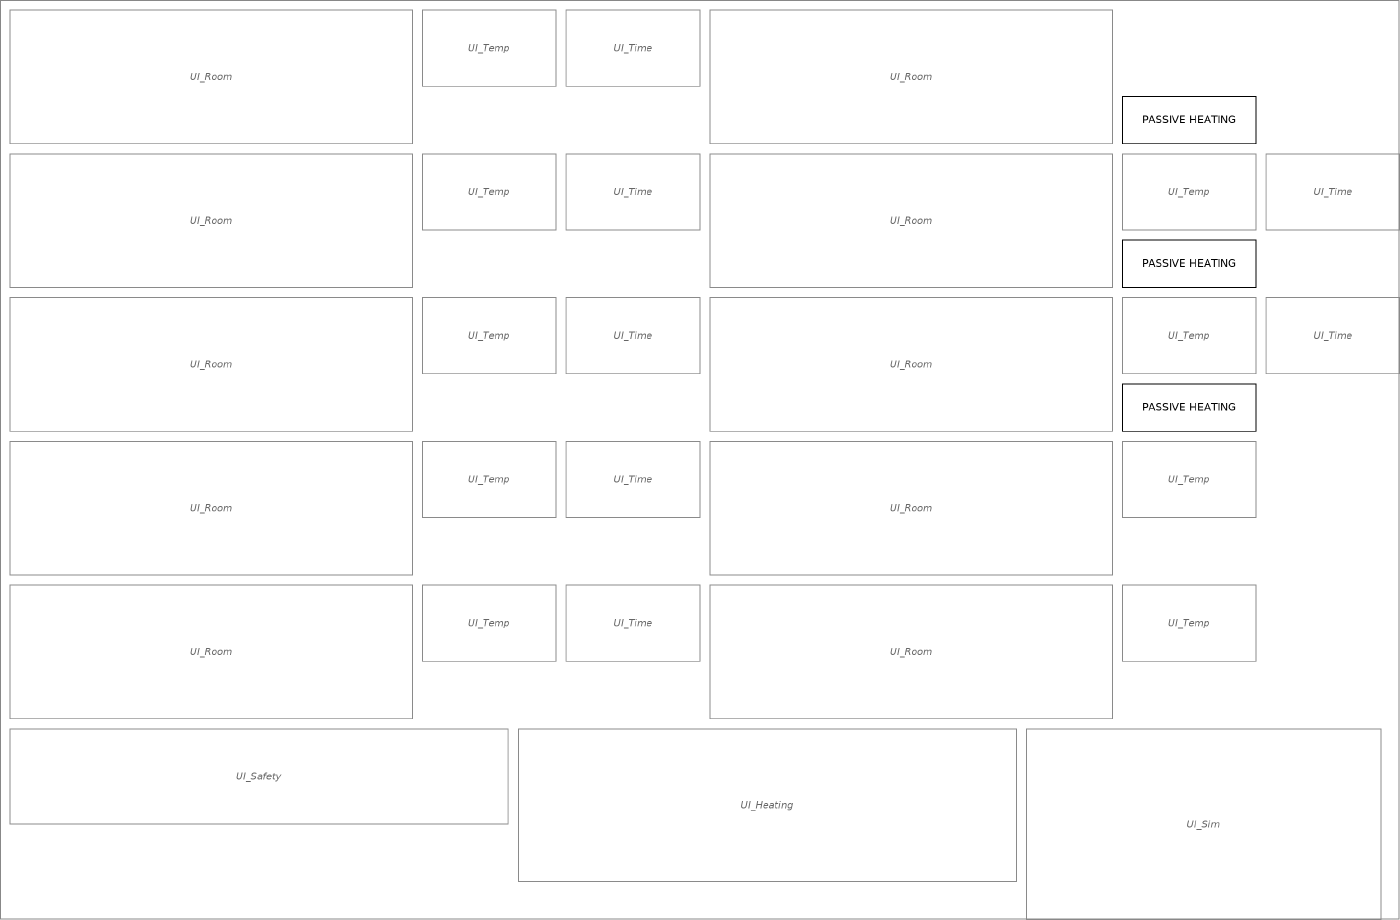
VISUALIZATION MAIN  // 1460x960
    Frame (10,760 520x100)
        shows UI_Safety(pou := MAIN.safety)
    Frame (540,760 520x160)
        shows UI_Heating(pou := MAIN.heating)
    Frame (10,10 420x140)
        shows UI_Room(ctx := MAIN.standardRoom[1]._ctx)
    Frame (10,160 420x140)
        shows UI_Room(ctx := MAIN.standardRoom[2]._ctx)
    Frame (10,310 420x140)
        shows UI_Room(ctx := MAIN.standardRoom[3]._ctx)
    Frame (10,460 420x140)
        shows UI_Room(ctx := MAIN.standardRoom[4]._ctx)
    Frame (10,610 420x140)
        shows UI_Room(ctx := MAIN.standardRoom[5]._ctx)
    Frame (440,10 140x80)
        shows UI_Temp(setting := MAIN.standardRoom[1]._settings.temp)
    Frame (440,160 140x80)
        shows UI_Temp(setting := MAIN.standardRoom[2]._settings.temp)
    Frame (440,310 140x80)
        shows UI_Temp(setting := MAIN.standardRoom[3]._settings.temp)
    Frame (440,460 140x80)
        shows UI_Temp(setting := MAIN.standardRoom[4]._settings.temp)
    Frame (440,610 140x80)
        shows UI_Temp(setting := MAIN.standardRoom[5]._settings.temp)
    Frame (740,10 420x140)
        shows UI_Room(ctx := MAIN.receptionRoom._ctx)
    Frame (740,160 420x140)
        shows UI_Room(ctx := MAIN.conferentionRoom01._ctx)
    Frame (740,310 420x140)
        shows UI_Room(ctx := MAIN.conferentionRoom02._ctx)
    Frame (740,460 420x140)
        shows UI_Room(ctx := MAIN.storeRoom01._ctx)
    Frame (740,610 420x140)
        shows UI_Room(ctx := MAIN.storeRoom02._ctx)
    Frame (1170,160 140x80)
        shows UI_Temp(setting := MAIN.conferentionRoom01._settings.temp)
    Frame (1170,310 140x80)
        shows UI_Temp(setting := MAIN.conferentionRoom02._settings.temp)
    Frame (1170,460 140x80)
        shows UI_Temp(setting := MAIN.storeRoom01._settings)
    Frame (1170,610 140x80)
        shows UI_Temp(setting := MAIN.storeRoom02._settings)
    Frame (1320,160 140x80)
        shows UI_Time(settings := MAIN.conferentionRoom01._settings.timee)
    Frame (590,10 140x80)
        shows UI_Time(settings := MAIN.standardRoom[1]._settings.timee)
    Frame (590,160 140x80)
        shows UI_Time(settings := MAIN.standardRoom[2]._settings.timee)
    Frame (590,310 140x80)
        shows UI_Time(settings := MAIN.standardRoom[3]._settings.timee)
    Frame (590,610 140x80)
        shows UI_Time(settings := MAIN.standardRoom[5]._settings.timee)
    Frame (590,460 140x80)
        shows UI_Time(settings := MAIN.standardRoom[4]._settings.timee)
    Frame (1320,310 140x80)
        shows UI_Time(settings := MAIN.conferentionRoom02._settings.timee)
    Rectangle (1170,400 140x50), "PASSIVE HEATING", colour toggle: MAIN.conferentionRoom02._settings.bEnablePassive
        toggle MAIN.conferentionRoom02._settings.bEnablePassive
    Rectangle (1170,250 140x50), "PASSIVE HEATING", colour toggle: MAIN.conferentionRoom01._settings.bEnablePassive
        toggle MAIN.conferentionRoom01._settings.bEnablePassive
    Rectangle (1170,100 140x50), "PASSIVE HEATING"
        toggle MAIN.receptionRoom._bEnablePassive
    Frame (1070,760 370x200)
        shows UI_Sim(param := SIM.param)
END_VISUALIZATION

(* stored: Version 1.1.0.1
   Visu MAIN: Id {1e026e4d-f1dc-41ee-aecc-8d5674db4a1b} *)
